FUNCTION TryConvert_USINT_TO_BYTE : BOOL
VAR_INPUT
	in : USINT;
	out : REFERENCE TO BYTE;
END_VAR

out := USINT_TO_BYTE(in);
TryConvert_USINT_TO_BYTE := TRUE;

END_FUNCTION

(* stored: Version 1.1.0.1, ProductVersion 3.1.4024.12
   POU TryConvert_USINT_TO_BYTE: Id {ef7b5d3d-1892-44e3-8b42-45254579f1b6}, SpecialFunc None *)
